INTERFACE I_HE_SATT_Sequence

METHOD Start
VAR_INPUT
    fRequestedAttenuation : LREAL; // [0.0 - 1.0]
END_VAR
END_METHOD

END_INTERFACE

(* stored: Version 1.1.0.1
   Itf I_HE_SATT_Sequence: Id {0db00903-e467-4eba-a2ac-5c1710fe2d80}
   Method Start: Id {e0b04e5d-646a-4a8b-b8e5-a82e75dd5e38} *)
